INTERFACE I_UniversalAxis_1

PROPERTY Acceleration : LREAL
GET
END_GET
SET
END_SET
END_PROPERTY

PROPERTY Active : REFERENCE TO BOOL
GET
END_GET
END_PROPERTY

PROPERTY ActualPosition : REFERENCE TO LREAL
GET
END_GET
END_PROPERTY

PROPERTY ActualVelocity : REFERENCE TO LREAL
GET
END_GET
END_PROPERTY

PROPERTY AxisRef : AXIS_REF
GET
END_GET
SET
END_SET
END_PROPERTY

PROPERTY BufferMode : MC_BufferMode
GET
END_GET
SET
END_SET
END_PROPERTY

PROPERTY Busy : REFERENCE TO BOOL
GET
END_GET
END_PROPERTY

PROPERTY Deceleration : LREAL
GET
END_GET
SET
END_SET
END_PROPERTY

PROPERTY Direction : Tc2_MC2.MC_Direction
GET
END_GET
SET
END_SET
END_PROPERTY

PROPERTY Error : REFERENCE TO BOOL
GET
END_GET
END_PROPERTY

PROPERTY ErrorID : REFERENCE TO UDINT
GET
END_GET
END_PROPERTY

PROPERTY HaltedCA : REFERENCE TO BOOL
GET
END_GET
END_PROPERTY

PROPERTY InPosition : REFERENCE TO BOOL
GET
END_GET
END_PROPERTY

PROPERTY InVelocity : REFERENCE TO BOOL
GET
END_GET
END_PROPERTY

PROPERTY IsHomed : REFERENCE TO BOOL
GET
END_GET
END_PROPERTY

PROPERTY Jerk : LREAL
GET
END_GET
SET
END_SET
END_PROPERTY

PROPERTY JogAcceleration : LREAL
GET
END_GET
SET
END_SET
END_PROPERTY

PROPERTY JogDeceleration : LREAL
GET
END_GET
SET
END_SET
END_PROPERTY

PROPERTY JogDirection : E_AxisJogDirection
GET
END_GET
SET
END_SET
END_PROPERTY

PROPERTY JogDone : REFERENCE TO BOOL
GET
END_GET
END_PROPERTY

PROPERTY JogJerk : LREAL
GET
END_GET
SET
END_SET
END_PROPERTY

PROPERTY JogMode : E_JogMode
GET
END_GET
SET
END_SET
END_PROPERTY

PROPERTY JogPosition : LREAL
GET
END_GET
SET
END_SET
END_PROPERTY

PROPERTY JogVelocity : LREAL
GET
END_GET
SET
END_SET
END_PROPERTY

PROPERTY LagError : LREAL
GET
END_GET
END_PROPERTY

PROPERTY MoveActive : REFERENCE TO BOOL
GET
END_GET
END_PROPERTY

METHOD MR_Abort : BOOL
END_METHOD

METHOD MR_FirstCycle
VAR_INPUT
	sName 				: STRING; 	(* Axis object name *)
	sMeasurementUnits	: STRING;	(* Measurement units used by axis *)
	bModulo				: BOOL;		(* Axis is periodic *)
END_VAR
END_METHOD

METHOD MR_Halt : BOOL
END_METHOD

METHOD MR_Home : BOOL
VAR_INPUT
	lrHomePosition : LREAL;
END_VAR
END_METHOD

METHOD MR_Init : BOOL
END_METHOD

METHOD MR_Jog : BOOL
VAR_INPUT
	//lrJogPosition : LREAL;
	//eJogDirection : E_AxisJogDirection;
	//eJogMode	  : E_JogMode;
	bJogActive	  : BOOL;
END_VAR
END_METHOD

METHOD MR_MoveAbsolute : BOOL
VAR_INPUT
	lrAbsolutePosition : LREAL;
END_VAR
END_METHOD

METHOD MR_MoveAdditive : BOOL
VAR_INPUT
	lrRelativeDistance : LREAL;
END_VAR
END_METHOD

METHOD MR_MoveRelative : BOOL
VAR_INPUT
	lrRelativeDistance : LREAL;
END_VAR
END_METHOD

METHOD MR_MoveVelocity : BOOL
END_METHOD

METHOD MR_Reset : BOOL
END_METHOD

METHOD MR_Stop : BOOL
END_METHOD

PROPERTY Name : STRING
GET
END_GET
SET
END_SET
END_PROPERTY

PROPERTY Options : ST_MoveOptions
GET
END_GET
SET
END_SET
END_PROPERTY

PROPERTY Override : LREAL
GET
END_GET
SET
END_SET
END_PROPERTY

PROPERTY PowerOn : REFERENCE TO BOOL
GET
END_GET
END_PROPERTY

PROPERTY ResetDone : REFERENCE TO BOOL
GET
END_GET
END_PROPERTY

PROPERTY SetpointPosition : LREAL
GET
END_GET
END_PROPERTY

PROPERTY SetpointVelocity : LREAL
GET
END_GET
END_PROPERTY

PROPERTY State : REFERENCE TO E_AxisState
GET
END_GET
END_PROPERTY

PROPERTY StatePlcOpen : REFERENCE TO E_AxisStatePlcOpen
GET
END_GET
END_PROPERTY

PROPERTY StopDeceleration : LREAL
GET
END_GET
SET
END_SET
END_PROPERTY

PROPERTY StopJerk : LREAL
GET
END_GET
SET
END_SET
END_PROPERTY

PROPERTY Stopped : REFERENCE TO BOOL
GET
END_GET
END_PROPERTY

PROPERTY Unit : STRING
GET
END_GET
SET
END_SET
END_PROPERTY

PROPERTY Velocity : LREAL
GET
END_GET
SET
END_SET
END_PROPERTY

END_INTERFACE

(* stored: Version 1.1.0.1, ProductVersion 3.1.4024.12
   Itf I_UniversalAxis_1: Id {94073e32-4de7-460c-b3e7-b8a11f6c7abd}
   Property Acceleration: Id {10065ca7-38cb-431a-967b-321f67ceac7e}
   Get Get: Id {0657e62a-daba-4f7f-81b7-87eb8a967ada}
   Set Set: Id {72de5533-4c74-4a0d-8848-1edc235943b5}
   Property Active: Id {d44ea5ed-6543-411d-97d2-78cd72d0e2a5}
   Get Get: Id {b5e21b9c-1d2f-4e88-8216-ce9cf6f5923c}
   Property ActualPosition: Id {adcf5a37-a6e6-45fd-a6b8-6c557668c82f}
   Get Get: Id {17777f09-0f59-45ae-9048-08a387883716}
   Property ActualVelocity: Id {19e3c654-ea4a-4e31-9835-bf9e303eb3cb}
   Get Get: Id {b77bbd2e-3528-42c1-870e-d8b08c5db19e}
   Property AxisRef: Id {99fff1fa-cd8f-4c59-ae72-2785d8953d02}
   Get Get: Id {43b64e1f-a2af-4bfa-a931-e1b5f3a40ad1}
   Set Set: Id {7a78a9b1-4c98-400b-8485-93edacdbc69d}
   Property BufferMode: Id {f860458e-07d6-4978-8fc3-9f9854ee1c00}
   Get Get: Id {c2c0c7ed-2eb5-444f-8430-ff8c9c5d94be}
   Set Set: Id {f040818d-34fc-4e21-a618-ebf9d7757e8e}
   Property Busy: Id {d77137f3-25fe-4d1f-af05-b80c1d4e312d}
   Get Get: Id {1992ff03-262c-4222-a4ba-1027628c8101}
   Property Deceleration: Id {608d22f5-c08e-4d68-bb74-49d0fa6711c3}
   Get Get: Id {a2ede01d-ce0d-4df4-a8cd-40bde7b0c6dc}
   Set Set: Id {f3736a91-fcdd-4705-a001-e16d6adb4c31}
   Property Direction: Id {1f57aba5-7680-4452-a01f-8b0467aa31c8}
   Get Get: Id {ae1ad5dc-b5d3-4e96-b35f-bf3816317d41}
   Set Set: Id {4124647b-420d-4f4f-9d34-c2e29f221dcb}
   Property Error: Id {6d3a33bf-3cf3-4eff-9ff9-fba2827723d4}
   Get Get: Id {a5fbec37-8b1a-4dd4-b1a2-4a21cd520e0c}
   Property ErrorID: Id {5018059c-9d71-448c-b2bc-70a1e1884e84}
   Get Get: Id {83da67e7-1672-47f7-ac93-413c77b5aa7e}
   Property HaltedCA: Id {2c399f20-de05-4f82-a3b5-4cfe1c1ef3c7}
   Get Get: Id {df5e1375-1765-4399-950c-7a52e57f74ba}
   Property InPosition: Id {9fa5572a-06fd-4332-ac3f-9d743ee500f1}
   Get Get: Id {8de0f21f-a41b-45f8-acf2-aa565faf8433}
   Property InVelocity: Id {bfe55979-1354-4cbc-b1b4-24d47ca368c0}
   Get Get: Id {cdc26b52-dd29-4731-9361-901546da620a}
   Property IsHomed: Id {855a07cb-c1a9-4e28-969c-89da2dde52c8}
   Get Get: Id {68b7b6f8-f996-4ee6-b54c-2b81af5cb83a}
   Property Jerk: Id {23136bdf-2a81-4150-8d40-0626452260f1}
   Get Get: Id {ee5c21ce-98aa-4b97-8b4c-63d46190f291}
   Set Set: Id {a3cd5de4-29b6-4e71-b3a8-ab0f065aefe5}
   Property JogAcceleration: Id {f9a40310-e830-4a06-ad29-cbcb9ea8cef1}
   Get Get: Id {d0399815-7d4b-4343-b22c-870dd250c267}
   Set Set: Id {b399536f-83ed-4693-9488-0b8d05fb5588}
   Property JogDeceleration: Id {eceae72f-5bc6-4fcc-881d-708f5923d062}
   Get Get: Id {28bca398-e3ff-42c3-9715-776acee10732}
   Set Set: Id {2ab8ab5a-72e3-49ad-afa6-3aceea6a07c9}
   Property JogDirection: Id {1ea946b2-3693-4091-9f66-520b8b5f5d82}
   Get Get: Id {121ded6f-6001-45b5-bca8-afe910de1b3e}
   Set Set: Id {d77d4ada-eb4c-44dd-914f-4b372fd631a2}
   Property JogDone: Id {e9d391ef-54e1-4edc-a168-8938f3f9ff98}
   Get Get: Id {c86af12d-4912-468c-957e-33ca6056590c}
   Property JogJerk: Id {416a156e-03a9-41b5-b8c1-af5e5d4f6ed6}
   Get Get: Id {779f9289-6be5-4a66-9353-43acd1f9ea41}
   Set Set: Id {c81d91eb-062c-4171-8185-6c726e836fe1}
   Property JogMode: Id {09591936-0362-4817-b12d-a41bbcfe1c65}
   Get Get: Id {e801d2fb-1e74-4007-af5c-c6207ecae62f}
   Set Set: Id {3cdcdb5d-4b9b-4835-a507-276b51db8823}
   Property JogPosition: Id {6520f860-2f70-4b41-87e7-683ae3a5b1e1}
   Get Get: Id {c1848c02-eb58-4c85-b234-f9e0c98ec93a}
   Set Set: Id {c3e57ae8-936a-41ca-a1bd-cd6426561300}
   Property JogVelocity: Id {ffa37301-d41b-40a7-9003-0ab1497e1f40}
   Get Get: Id {311c83d5-5dae-4cca-bf81-08dadee08eb6}
   Set Set: Id {8b3ffd50-264d-42f2-a41f-f9c0c04e9e3d}
   Property LagError: Id {9e867027-e80e-4a90-bd45-c386cd423e9d}
   Get Get: Id {0afd0e13-6100-44fc-bfa0-c036825ca4e5}
   Property MoveActive: Id {2b080632-b32e-4c4d-b764-ad5393cf7851}
   Get Get: Id {57eb4340-23c8-499b-a592-873dc894038b}
   Method MR_Abort: Id {e184fe4a-756f-42a8-b65a-1a9d93fed163}
   Method MR_FirstCycle: Id {8ef05237-bbb4-4d07-9bd3-f6e6e7baf26b}
   Method MR_Halt: Id {41900d55-4796-4419-9daa-69c1983bfd50}
   Method MR_Home: Id {78a3f703-bf3e-4426-81c2-c1c17627feb7}
   Method MR_Init: Id {c72a09f6-b7a0-4c4c-b390-29a3b8608bc9}
   Method MR_Jog: Id {8fe03705-f98c-4488-bd98-cb765dcc5461}
   Method MR_MoveAbsolute: Id {24c3ee15-3778-4429-92b6-14428b5bd29f}
   Method MR_MoveAdditive: Id {373c91d0-316a-469f-b002-d7db5368da36}
   Method MR_MoveRelative: Id {2b9cdef0-4063-4da1-8cb8-6b0975489d9a}
   Method MR_MoveVelocity: Id {519a80f0-b4b7-4d7c-8b9e-ac5214566d9f}
   Method MR_Reset: Id {292f1098-64cf-4760-b433-a3c271634443}
   Method MR_Stop: Id {4d593337-6b5f-4013-a4cb-af7797de0fa7}
   Property Name: Id {dc34c785-d010-4bdc-9b19-5facb87bd8e7}
   Get Get: Id {a752c9fe-f1b9-448a-953e-ae319bc39bd5}
   Set Set: Id {0cd42eef-bab9-4f40-9a24-9552b6d3b2b9}
   Property Options: Id {ce07fd8a-d41a-4b93-b780-f83931ca31b2}
   Get Get: Id {9a45c83c-057d-4189-9bdb-45e8ef57b79c}
   Set Set: Id {a022051e-4f9d-4f37-9b65-8b004131d00c}
   Property Override: Id {729530af-1459-4f45-9b40-bd7b233c4219}
   Get Get: Id {da133db4-7539-461d-a1f7-b05a79426327}
   Set Set: Id {22e0df87-ed29-4c0f-8f27-413a34578c62}
   Property PowerOn: Id {0e2f8b24-4d62-4135-937e-d06fc010a5e3}
   Get Get: Id {f817c9b4-420c-49d5-bb85-83f5c652858e}
   Property ResetDone: Id {2f36091d-3124-4aa7-927a-bf7a2e93169b}
   Get Get: Id {0f320a23-bdea-4a20-a298-5964d25b32e7}
   Property SetpointPosition: Id {feacd13b-80d5-4ad8-bc2d-cfa6df99cb46}
   Get Get: Id {9355baec-3d30-4373-bbcf-dfbcc5dd7088}
   Property SetpointVelocity: Id {785cc53f-f775-4491-8a55-6d4d8570f32b}
   Get Get: Id {3ebad751-a4f5-4c6e-9062-d68b06204aa6}
   Property State: Id {ed7d8797-0bfb-4dea-b6d3-aab4014c511d}
   Get Get: Id {83f1b559-2854-47b2-a30f-89120e71a979}
   Property StatePlcOpen: Id {e1d0ba81-0d72-4b69-bb68-8812957c07cb}
   Get Get: Id {13e08810-26fb-4cdf-bd11-269080ab01b4}
   Property StopDeceleration: Id {74d39688-4bc3-446a-a62d-ef69a9af5dd5}
   Get Get: Id {a56b1882-bc37-4b75-890b-3e5a0dbf52bf}
   Set Set: Id {b8afaf66-c543-4fdf-bd82-3e2c0bc2db85}
   Property StopJerk: Id {c9bf64a0-858f-4e3b-9e94-b328140cc7d7}
   Get Get: Id {8c362337-7320-4f30-b71b-d4ff90c1e733}
   Set Set: Id {01952ad1-c0f7-48bd-b6a9-af20feb30dfb}
   Property Stopped: Id {cd7a824d-6466-4aaf-a0aa-6c910b39668f}
   Get Get: Id {e2e9f82b-3d75-45f2-8b4d-8b432933fb25}
   Property Unit: Id {5d1d98c3-329e-489d-80ee-29d33a421073}
   Get Get: Id {3c1db143-7603-4d3b-b7a5-d7241ba954e0}
   Set Set: Id {90006c40-379f-451e-9bfd-f8c64a507dc5}
   Property Velocity: Id {8de0e14b-d46a-4690-a574-703fadd813ec}
   Get Get: Id {3f7d677c-4e79-4282-a076-7ddc7264f022}
   Set Set: Id {d8611525-c5dc-4790-88a8-cc6d24ba2445} *)
